// TIA Portal V20 export
TYPE "LKinCtrl_PathEditor_typeInternalEvents"
// stored: Access Published
   STRUCT
      addChangeCommand { ExternalAccessible := 'False'; ExternalVisible := 'False'; ExternalWritable := 'False'} : Struct
         trigger : Bool;
         mode : USInt;
         programNo : DInt;
         commandNo : DInt;
         command : "LKinCtrl_typePathDataElement";
      END_STRUCT;
   END_STRUCT;
END_TYPE
